(* IEC 61131-3 sources: Structured-Text/Source Code/Logic/TON_Pausable, 2 files *)

(* ---- Local Variables.ST ---- *)
VAR_INPUT
	IN: BOOL;
	PT: TIME;
	PAUSE: BOOL
END_VAR

VAR_OUTPUT
	Q: BOOL;
	ET: TIME;
END_VAR

VAR
	rtPause: R_TRIG;
	tTimePaused: TIME;
	Ton_A: TON;
	bTimedOut: BOOL;		//Prevents Ton_A.Q from resetting if paused when timed out.
END_VAR

(* ---- TON_Pausable.ST ---- *)
//Timer start Input Off, reset variables.;
IF NOT IN THEN
	tTimePaused := T#0s;
	bTimedOut := False;
END_IF;

//Check for pause input, store ET at time of pause.
//rtPause(CLK := PAUSE);
rtPause(PAUSE);
IF rtPause.Q THEN
    tTimePaused := tTimePaused + Ton_A.ET;
END_IF;

//Timer Definition.
Ton_A(IN := IN AND NOT PAUSE, PT := PT - tTimePaused);

//Output States.
IF Ton_A.Q THEN
	bTimedOut := TRUE;
END_IF;
Q := bTimedOut;
ET := tTimePaused + Ton_A.ET;
